{region '#Template'}
	{attribute 'Version' := '1.0.0.0'}
	{attribute 'Tags' := '"LCID": "1031", "Text": "GVL, DPAD, Trades, ObjectName, Description"'}
	{attribute 'Tags' := '"LCID": "1033", "Text": "GVL, DPAD, Trades, ObjectName, Description"'}
	{attribute 'Description' := '"LCID": "1031", "Text": "Textliste Gewerke"'}
	{attribute 'Description' := '"LCID": "1033", "Text": "Text list trades"'}
{endregion}

{attribute 'global_init_slot' := '40510'}
VAR_GLOBAL
  TxtTrade_Doors_gates_windows_sun_protection_sObjectName                :T_BA_StateText:='TTF';
  TxtTrade_Doors_gates_windows_sun_protection_sDescription                :T_BA_StateText:='Türen, Tore, Fenster, Sonnenschutz';
  TxtTrade_Sewage_water_and_gas_plants_sObjectName                       :T_BA_StateText:='GWA';
  TxtTrade_Sewage_water_and_gas_plants_sDescription                       :T_BA_StateText:='Abwasser-, Wasser-, Gasanlagen';
  TxtTrade_Heat_supply_systems_sObjectName                               :T_BA_StateText:='HZG';
  TxtTrade_Heat_supply_systems_sDescription                               :T_BA_StateText:='Wärmeversorgungsanlagen';
  TxtTrade_Air_conditioning_sObjectName                                  :T_BA_StateText:='LTA';
  TxtTrade_Air_conditioning_sDescription                                  :T_BA_StateText:='Lufttechnische Anlagen';
  TxtTrade_Refrigeration_systems_sObjectName                             :T_BA_StateText:='KAE';
  TxtTrade_Refrigeration_systems_sDescription                             :T_BA_StateText:='Kälteanlagen';
  TxtTrade_High_voltage_systems_sObjectName                              :T_BA_StateText:='ELT';
  TxtTrade_High_voltage_systems_sDescription                              :T_BA_StateText:='Starkstromanlagen';
  TxtTrade_Telecommunication_and_information_technology_sObjectName      :T_BA_StateText:='FIA';
  TxtTrade_Telecommunication_and_information_technology_sDescription      :T_BA_StateText:='Fernm.- und informationstech. Anlagen';
  TxtTrade_Hazard_detection_and_alarm_systems_sObjectName                :T_BA_StateText:='GMA';
  TxtTrade_Hazard_detection_and_alarm_systems_sDescription                :T_BA_StateText:='Gefahrenmelde- und Alarmanlagen';
  TxtTrade_Conveyors_sObjectName                                         :T_BA_StateText:='FTA';
  TxtTrade_Conveyors_sDescription                                         :T_BA_StateText:='Förderanlagen';
  TxtTrade_Kitchen_technology_systems_sObjectName                        :T_BA_StateText:='KTA';
  TxtTrade_Kitchen_technology_systems_sDescription                        :T_BA_StateText:='Küchentechnische Anlagen';
  TxtTrade_Laundry_and_cleaning_systems_sObjectName                      :T_BA_StateText:='WAR';
  TxtTrade_Laundry_and_cleaning_systems_sDescription                      :T_BA_StateText:='Wäscherei- und Reinigungsanlagen';
  TxtTrade_Media_supply_systems_sObjectName                              :T_BA_StateText:='MVA';
  TxtTrade_Media_supply_systems_sDescription                              :T_BA_StateText:='Medienversorgungsanlagen';
  TxtTrade_Medical_and_laboratory_equipment_sObjectName                  :T_BA_StateText:='MED';
  TxtTrade_Medical_and_laboratory_equipment_sDescription                  :T_BA_StateText:='Medizin- und labortechnische Anlagen';
  TxtTrade_Fire_extinguishing_systems_sObjectName                        :T_BA_StateText:='FLA';
  TxtTrade_Fire_extinguishing_systems_sDescription                        :T_BA_StateText:='Feuerlöschanlagen';
  TxtTrade_Bathing_facilities_sObjectName                                :T_BA_StateText:='BTA';
  TxtTrade_Bathing_facilities_sDescription                                :T_BA_StateText:='Badetechnische Anlagen';
  TxtTrade_Process_heating_cooling_and_air_systems_sObjectName           :T_BA_StateText:='PRO';
  TxtTrade_Process_heating_cooling_and_air_systems_sDescription           :T_BA_StateText:='Prozesswärme-, -kälte- und -luftanlagen';
  TxtTrade_Waste_disposal_facilities_sObjectName                         :T_BA_StateText:='ENT';
  TxtTrade_Waste_disposal_facilities_sDescription                         :T_BA_StateText:='Entsorgungsanlagen';
  TxtTrade_Building_automation_and_control_systems_general_sObjectName   :T_BA_StateText:='GAS';
  TxtTrade_Building_automation_and_control_systems_general_sDescription   :T_BA_StateText:='Gebäudeautomation allgemein';
  TxtTrade_Automation_focal_point_information_focal_point_sObjectName    :T_BA_StateText:='ASP';
  TxtTrade_Automation_focal_point_information_focal_point_sDescription    :T_BA_StateText:='Automationsschwerpunkt';
  TxtTrade_Room_automation_sObjectName                                   :T_BA_StateText:='RAU';
  TxtTrade_Room_automation_sDescription                                   :T_BA_StateText:='Raumautomation';
  TxtTrade_Outdoor_devices_sObjectName                                   :T_BA_StateText:='AUG';
  TxtTrade_Outdoor_devices_sDescription                                   :T_BA_StateText:='Außengeräte';
END_VAR

(* stored: Version 1.1.0.1, ProductVersion 3.1.4024.9
   GVL TxtTrade_1031: Id {0123b405-fa16-4245-9a96-721d26c3871a} *)
